PROGRAM Axis01_Command
VAR
	Axis01: AXIS_REF;											//회전축
	Axis01_MC_Home: FB_HomeBeforeMoveAX8000;
	Axis01_MC_Power: MC_Power;
	Axis01_Status: MC_ReadStatus;
	Axis01_Position_Read: MC_ReadActualPosition;
	Axis01_Velocity_Read: MC_ReadActualVelocity;
	Axis01_Reset: MC_Reset;										//모터 알람 리셋
	Axis01_Stop: MC_Stop;										//모터 정지
	Axis01_Press_Move: MC_MoveAbsolute;
	Axis01_Home_Pos_Move: MC_MoveAbsolute;
	Axis01_Wait_Pos_Move: MC_MoveAbsolute;
	Axis01_Target_Pos_Move: MC_MoveAbsolute;
	Axis01_Work_End_Move: MC_MoveAbsolute;
	Axis01_Jog: MC_Jog;
	
	Always_ON	:	BOOL	:=TRUE	;//상시 ON
	Always_OFF	:	BOOL	:=FALSE	;//상시 OFF

	Home_Interlock			:	BOOL	;
	Home_Pos_Interlock		: 	BOOL	;
	Wait_Pos_Interlock		:	BOOL	;
	Target_Pos_Interlock	:	BOOL	;
	Work_End_POs_Interlock	:	BOOL	;
	Axis01_Calibration: MC_MoveAbsolute;
	Axis01_Maint_Move: MC_MoveAbsolute;
	Axis01_Tool_Change_Move: MC_MoveAbsolute;
	Axis01_Calibration_Move: MC_MoveAbsolute;
	Timer04: TON;
	keb_R: BOOL;
END_VAR
VAR // added by the converter: edge detectors and wires of the graphical bodies
    _rt1 : R_TRIG;
END_VAR

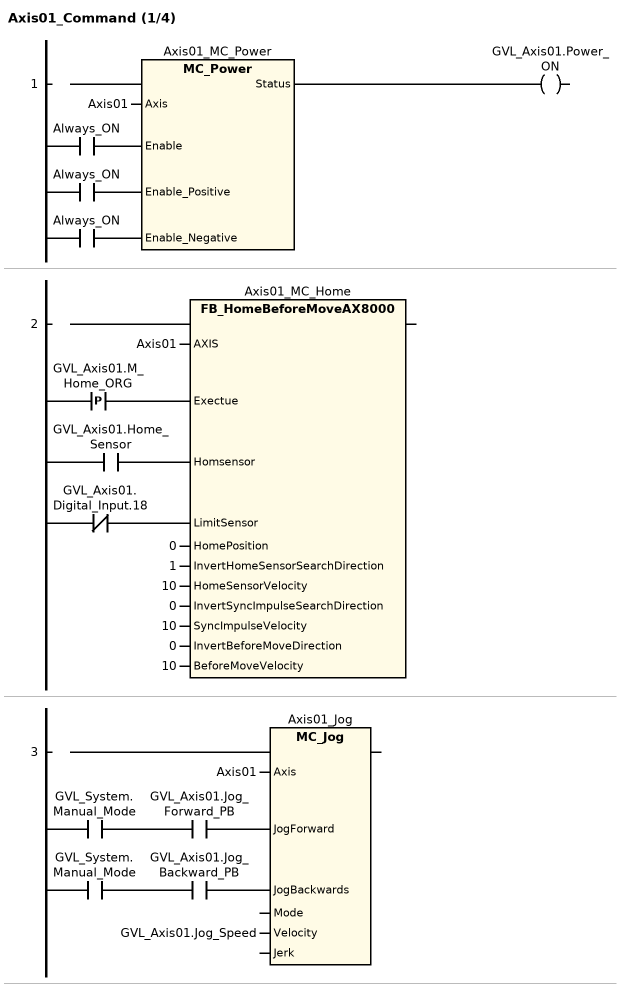
// NETWORK 1
Axis01_MC_Power(
    Axis := Axis01,
    Enable := Always_ON,
    Enable_Positive := Always_ON,
    Enable_Negative := Always_ON); // MC_Power
GVL_Axis01.Power_ON := Axis01_MC_Power.Status;

// NETWORK 2
_rt1(CLK := GVL_Axis01.M_Home_ORG);
Axis01_MC_Home(
    AXIS := Axis01,
    Exectue := _rt1.Q,
    Homsensor := GVL_Axis01.Home_Sensor,
    LimitSensor := NOT GVL_Axis01.Digital_Input.18,
    HomePosition := 0,
    InvertHomeSensorSearchDirection := 1,
    HomeSensorVelocity := 10,
    InvertSyncImpulseSearchDirection := 0,
    SyncImpulseVelocity := 10,
    InvertBeforeMoveDirection := 0,
    BeforeMoveVelocity := 10); // FB_HomeBeforeMoveAX8000

// NETWORK 3
Axis01_Jog(
    Axis := Axis01,
    JogForward := GVL_System.Manual_Mode AND GVL_Axis01.Jog_Forward_PB,
    JogBackwards := GVL_System.Manual_Mode AND GVL_Axis01.Jog_Backward_PB,
    Velocity := GVL_Axis01.Jog_Speed); // MC_Jog

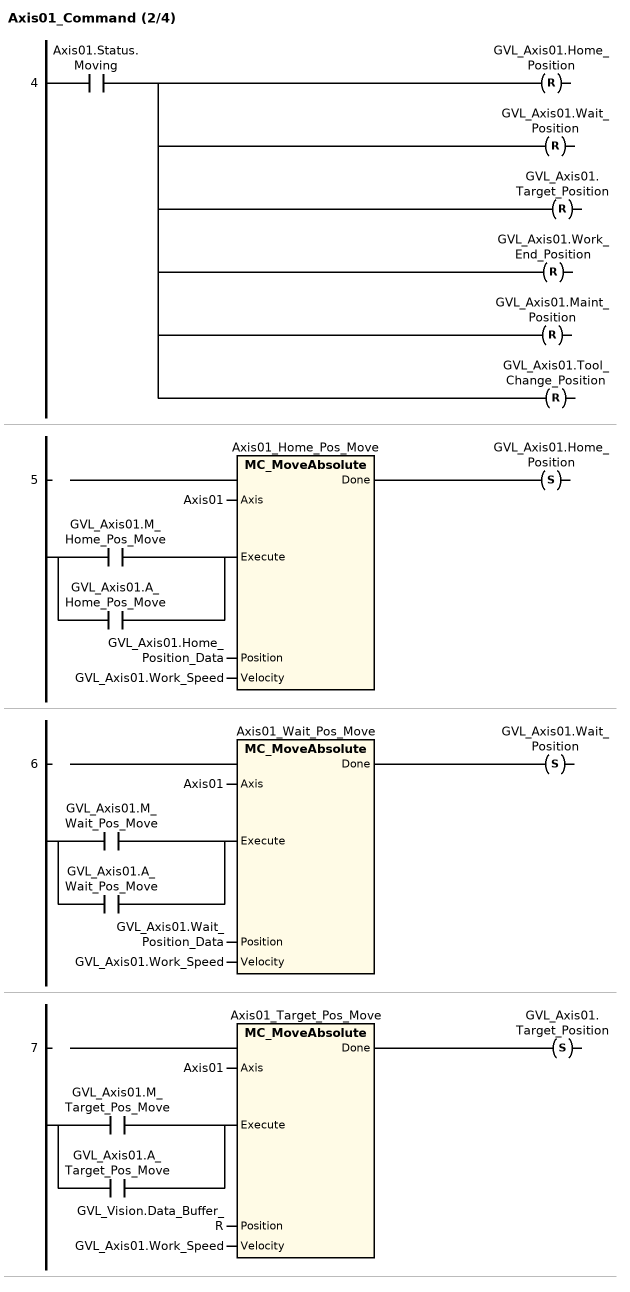
// NETWORK 4
GVL_Axis01.Home_Position R= Axis01.Status.Moving;
GVL_Axis01.Wait_Position R= Axis01.Status.Moving;
GVL_Axis01.Target_Position R= Axis01.Status.Moving;
GVL_Axis01.Work_End_Position R= Axis01.Status.Moving;
GVL_Axis01.Maint_Position R= Axis01.Status.Moving;
GVL_Axis01.Tool_Change_Position R= Axis01.Status.Moving;

// NETWORK 5
Axis01_Home_Pos_Move(
    Axis := Axis01,
    Execute := GVL_Axis01.M_Home_Pos_Move OR GVL_Axis01.A_Home_Pos_Move,
    Position := GVL_Axis01.Home_Position_Data,
    Velocity := GVL_Axis01.Work_Speed); // MC_MoveAbsolute
GVL_Axis01.Home_Position S= Axis01_Home_Pos_Move.Done;

// NETWORK 6
Axis01_Wait_Pos_Move(
    Axis := Axis01,
    Execute := GVL_Axis01.M_Wait_Pos_Move OR GVL_Axis01.A_Wait_Pos_Move,
    Position := GVL_Axis01.Wait_Position_Data,
    Velocity := GVL_Axis01.Work_Speed); // MC_MoveAbsolute
GVL_Axis01.Wait_Position S= Axis01_Wait_Pos_Move.Done;

// NETWORK 7
Axis01_Target_Pos_Move(
    Axis := Axis01,
    Execute := GVL_Axis01.M_Target_Pos_Move OR GVL_Axis01.A_Target_Pos_Move,
    Position := GVL_Vision.Data_Buffer_R,
    Velocity := GVL_Axis01.Work_Speed); // MC_MoveAbsolute
GVL_Axis01.Target_Position S= Axis01_Target_Pos_Move.Done;

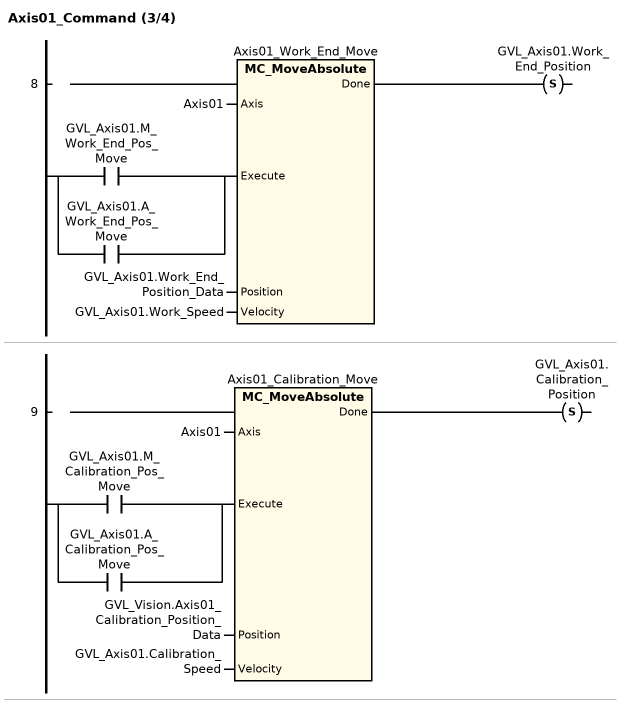
// NETWORK 8
Axis01_Work_End_Move(
    Axis := Axis01,
    Execute := GVL_Axis01.M_Work_End_Pos_Move OR GVL_Axis01.A_Work_End_Pos_Move,
    Position := GVL_Axis01.Work_End_Position_Data,
    Velocity := GVL_Axis01.Work_Speed); // MC_MoveAbsolute
GVL_Axis01.Work_End_Position S= Axis01_Work_End_Move.Done;

// NETWORK 9
Axis01_Calibration_Move(
    Axis := Axis01,
    Execute := GVL_Axis01.M_Calibration_Pos_Move OR GVL_Axis01.A_Calibration_Pos_Move,
    Position := GVL_Vision.Axis01_Calibration_Position_Data,
    Velocity := GVL_Axis01.Calibration_Speed); // MC_MoveAbsolute
GVL_Axis01.Calibration_Position S= Axis01_Calibration_Move.Done;

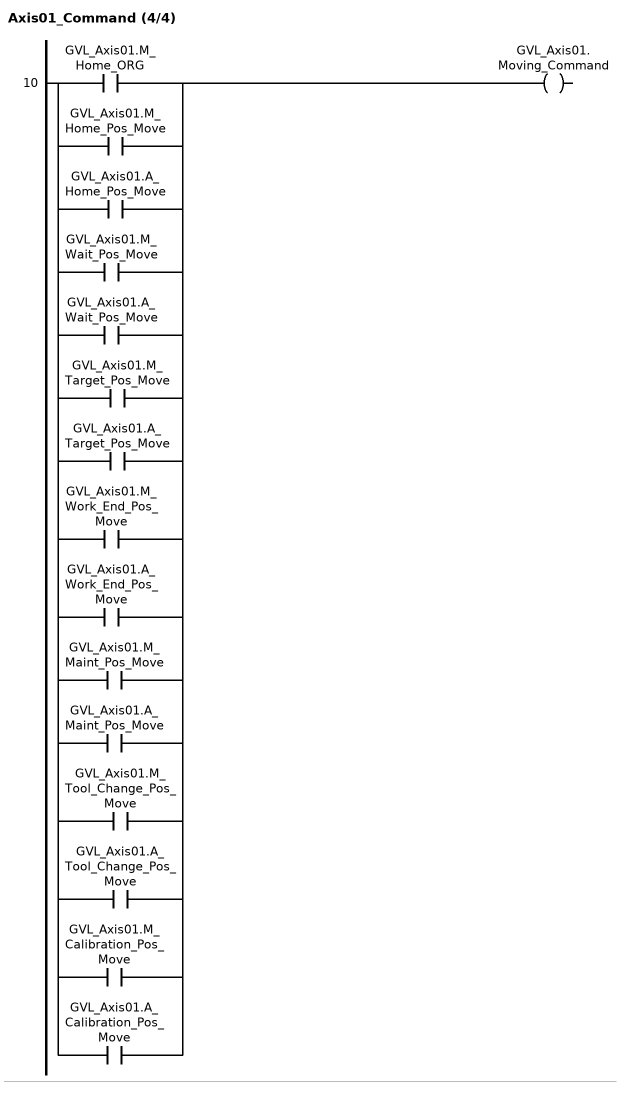
// NETWORK 10
GVL_Axis01.Moving_Command := GVL_Axis01.M_Home_ORG OR GVL_Axis01.M_Home_Pos_Move OR GVL_Axis01.A_Home_Pos_Move OR GVL_Axis01.M_Wait_Pos_Move OR GVL_Axis01.A_Wait_Pos_Move OR GVL_Axis01.M_Target_Pos_Move OR GVL_Axis01.A_Target_Pos_Move OR GVL_Axis01.M_Work_End_Pos_Move OR GVL_Axis01.A_Work_End_Pos_Move OR GVL_Axis01.M_Maint_Pos_Move OR GVL_Axis01.A_Maint_Pos_Move OR GVL_Axis01.M_Tool_Change_Pos_Move OR GVL_Axis01.A_Tool_Change_Pos_Move OR GVL_Axis01.M_Calibration_Pos_Move OR GVL_Axis01.A_Calibration_Pos_Move;

END_PROGRAM

(* stored: Version 1.1.0.1, ProductVersion 3.1.4024.16
   POU Axis01_Command: Id {65ca833e-3d91-4a54-92ba-775618f31e4d}, SpecialFunc None *)
